(* CoDeSys 2.3.9.37 project: Cap11_12.pro *)
(* Libraries: Standard.lib 4.10.05 12:14:46, IecSfc.lib 13.4.06 16:51:28 *)

(* Global variable list: Global_Variables *)
VAR_GLOBAL
      (* Entradas *)
	M: BOOL;
	X2: BOOL;
	Y2: BOOL;
	Y1: BOOL;
	X1: BOOL;
       (* Salidas *)
	arriba: BOOL;
	abajo: BOOL;
	izquierda: BOOL;
	derecha: BOOL;
       luz:BOOL;
END_VAR

(* POU PLC_PRG, CFC *)
PROGRAM PLC_PRG
VAR
END_VAR
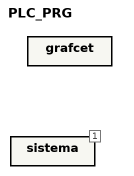
_CFC_ (* Continuous Function Chart, elements in execution order *)
#0 grafcet()
#1 sistema()
_END_CFC_
(* the same logic as Structured Text *)
grafcet();
sistema();
END_PROGRAM

(* POU grafcet, SFC *)
PROGRAM grafcet
VAR
END_VAR
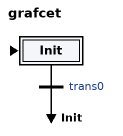
INITIAL_STEP Init:
END_STEP
TRANSITION FROM Init TO Init := trans0;
END_TRANSITION
END_PROGRAM

(* POU sistema, ST *)
PROGRAM sistema
VAR
  posx:REAL;
  posy:REAL;
	velx: REAL:=2;
	vely:REAL:=2;
  pertX:BOOL;
  pertY:BOOL;
END_VAR
IF arriba=TRUE THEN
   posy:=posy-vely;
END_IF

IF abajo=TRUE THEN
   posy:=posy+vely;
END_IF

IF derecha=TRUE THEN
   posx:=posx+velx;
END_IF

IF izquierda=TRUE THEN
   posx:=posx-velx;
END_IF

IF posx>515 AND posx<525 THEN
   Y2:=TRUE;
ELSE
   Y2:=FALSE;
END_IF

IF posx>-5 AND posx<5 THEN
   Y1:=TRUE;
ELSE
   Y1:=FALSE;
END_IF

IF posy<-295 AND posy>-305 THEN
   X2:=TRUE;
ELSE
   X2:=FALSE;
END_IF


IF posy>-5 AND posy<5 THEN
   X1:=TRUE;
ELSE
   X1:=FALSE;
END_IF


IF pertX=TRUE THEN
  posy:=posy+1;
END_IF

IF pertY=TRUE THEN
  posx:=posx+1;
END_IF
END_PROGRAM

(* Visualisation mesa
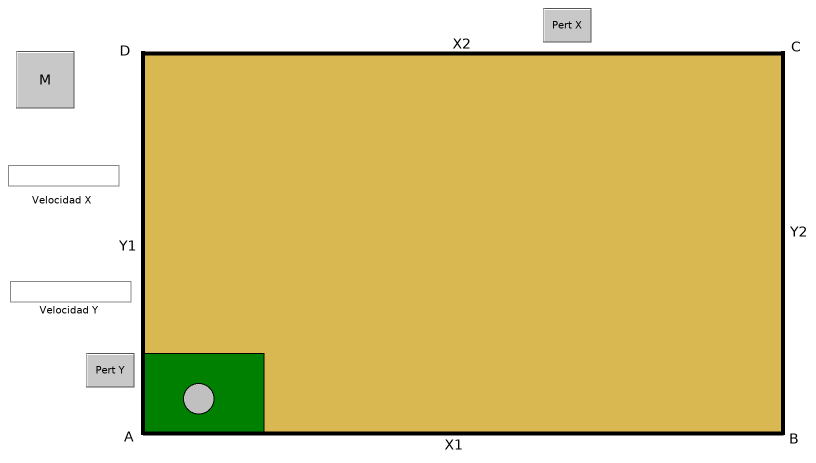
rectangle at (140,360)-(261,441): x offset sistema.posx; y offset sistema.posy
ellipse at (180,390)-(211,421): alarm colour if .luz; x offset sistema.posx; y offset sistema.posy
button at (13,58)-(71,115): text "M"; taps .M
polyline at (140,440)-(780,440): alarm colour if X1
polyline at (140,60)-(780,60): alarm colour if X2
polyline at (140,60)-(140,440): alarm colour if Y1
polyline at (780,60)-(780,440): alarm colour if Y2
rectangle at (104,427)-(148,460): text "A"
rectangle at (769,429)-(813,462): text "B"
rectangle at (771,37)-(815,70): text "C"
rectangle at (100,41)-(144,74): text "D"
rectangle at (437,34)-(481,67): text "X2"
rectangle at (429,435)-(473,468): text "X1"
rectangle at (774,222)-(818,255): text "Y2"
rectangle at (103,236)-(147,269): text "Y1"
rectangle at (14,188)-(104,226): text "Velocidad X"
rectangle at (21,298)-(111,336): text "Velocidad Y"
button at (540,15)-(588,49): text "Pert X"; taps sistema.pertX
button at (83,360)-(131,394): text "Pert Y"; taps sistema.pertY
3 more shapes without text or variables
*)
